FUNCTION_BLOCK TcoInspectionGroup EXTENDS TcoInspector IMPLEMENTS ITcoInspectionGroup, ITcoInspectionGroupAct
VAR
    {attribute 'hide'}
    _done                     : BOOL;				
    {attribute 'hide'}
    _done_PV                  : BOOL;				
    _overallResult            : TcoComprehensiveResult;
    _currentRunResult         : TcoComprehensiveResult;
    _inspections              : ARRAY[0..LAST_INSPECTION_INDEX] OF ULINT;
	_inspectionsEmpty         : ARRAY[0..LAST_INSPECTION_INDEX] OF ULINT;
    _inspectionIndex          : INT;
    _tierAct                  : TcoCore.TcoTier(THIS^);
    _normalizedAllowedRetries : UINT;
	
	
END_VAR

VAR CONSTANT
    LAST_INSPECTION_INDEX : INT := 50;
	MAX_NORMALIZED_RETRIES : UINT := 65535;
END_VAR

VAR 
	count : ULINT;
END_VAR

(*~
	<summary>
		Initiates grouped inspection.
	</summary>
~*)
METHOD Act : ITcoInspectionGroup
//VAR_IN_OUT
//	inoResult : TcoComprehensiveResult;
//END_VAR
OverInspected := FALSE;
_inspectionIndex          := 0;
_done                     := TRUE; // True then set to false if any inspector not done.
_normalizedAllowedRetries := MAX_NORMALIZED_RETRIES;
Act := THIS^;



IF (_tierAct.IsNewTier()) THEN
	_inspections:=_inspectionsEmpty;
    ClearResult(_currentRunResult);
END_IF
END_METHOD

METHOD ClearResult
VAR_IN_OUT
	inoResult : TcoComprehensiveResult;
END_VAR
inoResult.ErrorCodes := '';
inoResult.Failures := '';
inoResult.Result := eOverallResult.NoAction;
END_METHOD

(*~
	<docu>
		<summary>
			Gets common data settings of inspectors.
		</summary>			
	</docu>	
~*)
PROPERTY CommonData : REFERENCE TO TcoInspectorData
GET
VAR
	_data : TcoInspectorData; 
END_VAR
CommonData REF= _data;
END_GET
END_PROPERTY

METHOD Dialog : BOOL
VAR_INPUT
	inRetryStep : INT;
END_VAR
IF(THIS^.Done) THEN
	_tcoInspectorDialogue.OverInspected := THIS^.OverInspected;		
	IF(THIS^._currentRunResult.Result = eOverallResult.Failed) THEN
		THIS^._tcoInspectorDialogue.Invoke();
		_tcoInspectorDialogue();	
		
		{warning disable C0357}
		IF(_tcoInspectorDialogue._dialogRetry) THEN			
			Retry(inRetryStep);			
		END_IF
		
		IF(_tcoInspectorDialogue._dialogTerminate) THEN
			Terminate();
		END_IF
		
		IF(_tcoInspectorDialogue._dialogOverride) THEN
			CarryOn();
		END_IF
		{warning enable C0357}
	ELSE
		IF(Coordinator <> 0) THEN
			Coordinator.MoveNext();
		END_IF;	
	END_IF;	
END_IF;
END_METHOD

METHOD DialogWithExternalClose : BOOL
VAR_INPUT
	inRetryStep : INT;
	inRetrySignal:BOOL;
	inTerminateSignal : BOOL;
END_VAR
//IF THIS^._tcoInspectorDialogue.State=eTaskState.Ready THEN
//	THIS^._tcoInspectorDialogue.DialogRetry 	    :=  FALSE;	
//	THIS^._tcoInspectorDialogue.DialogTerminate  	:=  FALSE;	
//	THIS^._tcoInspectorDialogue.DialogOverride   	:=  FALSE;
//END_IF




_tcoInspectorDialogue.HandleExternalSignals(inRetrySignal:=inRetrySignal,inTerminateSignal:=inTerminateSignal);


IF(THIS^.Done) THEN
	_tcoInspectorDialogue.OverInspected := THIS^.OverInspected;		
	IF(THIS^._currentRunResult.Result = eOverallResult.Failed) THEN
		THIS^._tcoInspectorDialogue.Invoke();
		_tcoInspectorDialogue();	
						
		
		{warning disable C0357}
		IF(_tcoInspectorDialogue._dialogRetry AND _tcoInspectorDialogue.DialogIsClosed ) THEN			
			Retry(inRetryStep);	
	
		END_IF
		
		IF(_tcoInspectorDialogue._dialogTerminate AND _tcoInspectorDialogue.DialogIsClosed ) THEN
			Terminate();
		END_IF
		
		IF(_tcoInspectorDialogue._dialogOverride AND _tcoInspectorDialogue.DialogIsClosed) THEN
			CarryOn();
		END_IF
		{warning enable C0357}
	ELSE
		IF(Coordinator <> 0) THEN
			Coordinator.MoveNext();
		END_IF;	
	END_IF;	
END_IF;

IF THIS^._tcoInspectorDialogue.State=eTaskState.Done 
		AND ( _tcoInspectorDialogue.DialogRetry
		OR _tcoInspectorDialogue.DialogTerminate
		OR _tcoInspectorDialogue.DialogOverride)
		AND _tcoInspectorDialogue.DialogIsClosed  THEN	
	THIS^._tcoInspectorDialogue.Restore();
END_IF;
END_METHOD

PROPERTY Done : BOOL
GET
Done := _done;
END_GET
END_PROPERTY

(*~
	<docu>
		<summary>
			Upon failure the inspection retries given number of time. When it reach	given numbers then terminate 		
		</summary>			
	</docu>	
~*)

{attribute 'hide'}
{attribute 'obsolete' := 'You should access `Evaluate` method via `OnFail()` method.'}
METHOD PUBLIC Evaluate : BOOL
VAR_INPUT
    (*~
	<docu>
		<summary>
			State from which the inspection will restart.		
		</summary>			
	</docu>	
	~*)
    inFromState : INT;
    (*~
	<docu>
		<summary>
			Behavior when ispection is failed		
		</summary>			
	</docu>	
	~*)
    inFailMode : eTcoInspectorFailMode;
    (*~
	<docu>
		<summary>
			State from which the inspection will continue.		
		</summary>			
	</docu>	
	~*)
    inToState : INT;
END_VAR
IF (_coordinator = 0) THEN
    RETURN;
END_IF

IF (THIS^.Done) THEN
    IF (THIS^._currentRunResult.Result = eOverallResult.Failed) THEN
        IF (__ISVALIDREF(_refOverallResult)) THEN
            _refOverallResult := _originalOverallResult;
        END_IF

        IF inFailMode = eTcoInspectorFailMode.CarryOn THEN
            _coordinator.MoveNext();
        ELSIF inFailMode = eTcoInspectorFailMode.JumpTo THEN
            _coordinator.Retry(inToState);
        ELSIF inFailMode = eTcoInspectorFailMode.Terminate THEN
            _coordinator.Terminate();
        ELSIF inFailMode = eTcoInspectorFailMode.RetryThenCarryOn THEN
            IF OverInspected THEN
                _coordinator.MoveNext();
            ELSE
                _coordinator.Retry(inFromState);
            END_IF;
        ELSIF inFailMode = eTcoInspectorFailMode.RetryThenJumpTo THEN
            IF OverInspected THEN
                _coordinator.Retry(inToState);
            ELSE
                _coordinator.Retry(inFromState);
            END_IF;

        ELSIF inFailMode = eTcoInspectorFailMode.RetryThenTeminate THEN
            IF OverInspected THEN
                _coordinator.Terminate();
            ELSE
                _coordinator.Retry(inFromState);
            END_IF;

        END_IF
    ELSE

        _coordinator.MoveNext();
    END_IF;
END_IF;

Evaluate := THIS^.Done;
END_METHOD

(*~
	<summary>
		Add inspector to inspection group to inspect
	</summary>
~*)
METHOD Inspect : ITcoInspectionGroup
VAR_INPUT
    Inspector : IInspector;
END_VAR
OnEnterInspection();

IF(_normalizedAllowedRetries <> 0 
AND _normalizedAllowedRetries <> MAX_NORMALIZED_RETRIES) THEN
	Inspector.CommonData.NumberOfAllowedRetries := _normalizedAllowedRetries;
END_IF;

Inspect := THIS^;


IF(Inspector.OverInspected) THEN
	THIS^.OverInspected := TRUE;
END_IF;

IF (Inspector.Done) THEN
    Inspector.UpdateComprehensiveResult(_currentRunResult);							
ELSE
	_done := FALSE;	
	_done_PV := FALSE;	
END_IF


IF(_inspectionIndex < LAST_INSPECTION_INDEX)THEN
	_inspections[_inspectionIndex] :=  Inspector.Identity;
	_inspectionIndex := _inspectionIndex + 1;
END_IF
END_METHOD

(*~
	<summary>
		Sets lower `number of allowed retries` for this call of inspection group.
		Invoke this method multiple times if you want to check for the inspection for lowest numebr of retries.
		<note type="important">
			The inspections will run at least once before allowed entries is normalized.
		</note>
	</summary>
~*)

METHOD NormalizeRetries : ITcoInspectionGroup
VAR_INPUT
	inoInspection : IInspector;
END_VAR
// Determine lowest number of retries
NormalizeRetries := THIS^;
IF( inoInspection.CommonData.NumberOfAllowedRetries <> 0 
AND_THEN inoInspection.CommonData.NumberOfAllowedRetries < _normalizedAllowedRetries) THEN
	_normalizedAllowedRetries := inoInspection.CommonData.NumberOfAllowedRetries;
END_IF
END_METHOD

METHOD OnFail : IOnFail
VAR_INPUT
END_VAR
//THIS^._tcoInspectorDialogue.SetInspector(THIS^);
OnFail := THIS^;
END_METHOD

(*~
	<docu>
		<summary>
			Gets `true` when the number of inspections excceds `NumberOfAllowedRetries`.
		</summary>			
	</docu>	
~*)
PROPERTY PUBLIC OverInspected : BOOL
GET
OverInspected := _isOverInspected;
END_GET
SET
_isOverInspected := OverInspected;
END_SET
END_PROPERTY

{attribute 'hide'}
{attribute 'obsolete' := 'You should access `Retry` method via `OnFail()` method.'}
METHOD Retry : BOOL
VAR_INPUT
	inFromState : INT;
END_VAR
IF(_coordinator = 0) THEN
	RETURN;	
END_IF

IF(THIS^.Done) THEN
	IF(THIS^._currentRunResult.Result = eOverallResult.Failed) THEN		
		IF(__ISVALIDREF(_refOverallResult)) THEN
			_refOverallResult := _originalOverallResult;
		END_IF	 
		ClearResult(_currentRunResult);	   	
		_coordinator.Retry(inFromState);
	ELSE
		_coordinator.MoveNext();
	END_IF;	
END_IF;	


Retry := THIS^.Done;
END_METHOD

{attribute 'hide'}
{attribute 'obsolete' := 'You should access `RetryThenTerminate` method via `OnFail()` method.'}
METHOD RetryThenTerminate : BOOL
VAR_INPUT
	inFromState : INT;
END_VAR
IF (_coordinator = 0) THEN
    RETURN;
END_IF

IF (THIS^.Done) THEN
    IF (THIS^._currentRunResult.Result = eOverallResult.Failed) THEN
        IF (__ISVALIDREF(_refOverallResult)) THEN
            _refOverallResult := _originalOverallResult;
        END_IF

        ClearResult(_currentRunResult);
        IF OverInspected THEN
            _coordinator.Terminate();
        ELSE
            _coordinator.Retry(inFromState);
        END_IF;
    ELSE
        _coordinator.MoveNext();
    END_IF;
END_IF;

RetryThenTerminate := THIS^.Done;
END_METHOD

{attribute 'hide'}
{attribute 'obsolete' := 'You should access `Terminate` method via `OnFail()` method.'}
METHOD Terminate : BOOL
IF(_coordinator = 0) THEN
	RETURN;	
END_IF

IF(THIS^.Done) THEN
	IF(THIS^._currentRunResult.Result = eOverallResult.Failed) THEN
		_coordinator.Terminate();
	ELSE
		_coordinator.MoveNext();
	END_IF;	
END_IF;	

Terminate := THIS^.Done;
END_METHOD

(*~
	<docu>
		<summary>
			Updates comprehensive result. The comprehensive result is set to `Failed` when any inspection fails or is inconclusive.
			Any bypassed or excluded inspection are not taken in the account.			
		</summary>			
	</docu>	
~*)

METHOD UpdateComprehensiveResult : IInspector
VAR_IN_OUT
	(*~
	<docu>
		<summary>
			Comprehensive result data structure to be updated.	
		</summary>			
	</docu>	
	~*)
    inoResult : TcoComprehensiveResult;
END_VAR
UpdateComprehensiveResult := THIS^;

_refOverallResult REF= inoResult;

IF(_tierUpdateOverall.IsNewTier()) THEN	
	_originalOverallResult := inoResult;
END_IF

		
CASE _currentRunResult.Result OF
	eOverallResult.NoAction:
		;
	eOverallResult.Passed:
		;
	eOverallResult.Failed:
		 
		_refOverallResult.Result		:= eOverallResult.Failed;
		_refOverallResult.Failures		:= _currentRunResult.Failures;
		_refOverallResult.ErrorCodes	:= _currentRunResult.ErrorCodes;
END_CASE


IF(_done) THEN
	_overallResult := _refOverallResult;
END_IF;
END_METHOD

(*~
	<docu>
		<summary>
			Updates failure description. Adding `FailureDescription` do the overall result structure.
		</summary>	
	</docu>	
~*)
METHOD PROTECTED UpdateDescriptions
VAR_IN_OUT
	inoResult : TcoComprehensiveResult;
END_VAR
IF NOT _done THEN
	_done_PV := FALSE;	
END_IF
IF(_done AND NOT _done_PV) THEN
	inoResult.Failures := THIS^.Context.Environment.Messaging.StringBuilder.Clear()
				.Append(inoResult.Failures)				
				.Append(CommonData.FailureDescription)
				.Append(';')
				.ToString();
	
	inoResult.ErrorCodes := THIS^.Context.Environment.Messaging.StringBuilder.Clear()
				.Append(inoResult.ErrorCodes)				
				.Append(CommonData.ErrorCode)
				.Append(';')
				.ToString();			
	_done_PV := TRUE;	
END_IF;
END_METHOD

METHOD WithCoordinator : ITcoInspectionGroupAct
VAR_INPUT
	inCoordinator : TcoCore.ITcoCoordinator;
END_VAR
_WithCoordinator(inCoordinator);
WithCoordinator := THIS^;
END_METHOD

END_FUNCTION_BLOCK

(* stored: Version 1.1.0.1, ProductVersion 3.1.4024.12
   POU TcoInspectionGroup: Id {d3e13610-7815-0c15-1fa4-6b11279e6aa5}, SpecialFunc None
   Folder OnFail: Id {6587d444-c4c8-0ba3-0430-72f2e8ae8a7c}
   Method Act: Id {35f139a3-c8e1-0dfe-09ea-5e112c3b9b62}
   Method ClearResult: Id {f7b2a68e-e38b-05d5-0a30-07f805d8c74c}
   Property CommonData: Id {36a6e3dd-6add-0a42-3ea4-eeae0ddbf08c}
   Get Get: Id {cf4f926b-9654-03bf-18da-2882eac3e99a}
   Method Dialog: Id {74a2f6ff-2257-0b1f-0c44-f3b62d0819e8}
   Method DialogWithExternalClose: Id {672e39a2-df24-00dc-01ed-378f101e1a1c}
   Property Done: Id {5d8b674b-9e76-0be3-1a04-7b0897c7e892}
   Get Get: Id {11835c00-ed30-04c2-28e0-db016edb13b4}
   Method Evaluate: Id {ec0c8dd4-dd5c-0319-2bb9-6b847f04a479}
   Method Inspect: Id {5050b1c2-e64a-023f-2d54-61af21de371f}
   Method NormalizeRetries: Id {ded8cb66-c7fe-0d86-039b-c79bf8c6c339}
   Method OnFail: Id {ad5daf18-5adf-0409-3fbe-22acf686dffa}
   Property OverInspected: Id {e0f14d06-9cf8-02a2-1ed1-c4992364d32d}
   Get Get: Id {e3256b18-3d99-064d-3cee-3418b265bdcd}
   Set Set: Id {588b6ea8-8508-0f69-0956-a218a73d88ea}
   Method Retry: Id {35486965-61f5-0154-3790-1cbb7d6396ad}
   Method RetryThenTerminate: Id {a1d11a84-0c54-0300-27d8-3ee3e5fb3c1c}
   Method Terminate: Id {ef8afc1b-48c1-0d87-3e46-8fe826fdd29c}
   Method UpdateComprehensiveResult: Id {84f70c65-26b9-0040-3478-66f5894d8644}
   Method UpdateDescriptions: Id {7760290a-e8d0-0302-18a7-ce0b9abf0e99}
   Method WithCoordinator: Id {c31bd8b7-9661-0564-2449-159a318fede9} *)
